FUNCTION_BLOCK ExerciseF_P1
VAR_IN_OUT
	Parameters: GreenMasterBaseParameters;
END_VAR
VAR_INPUT
	EN: BOOL := TRUE;
	ForceExercise: BOOL;
END_VAR
VAR_OUTPUT
	Exercising: BOOL;
END_VAR
VAR
	ExerciseTimer: Timer;
	LocalTime: FB_LocalSystemTime;
	Elapsed: LINT;
	CurrentState: INT;
	StateTimer: TImer;
	DetectedDamperError: BOOL;
	FirstTime: BOOL := TRUE;
END_VAR

LocalTime(bEnable := TRUE);
ExerciseTimer(EN := EN);
Elapsed := ExerciseTimer.ElapsedTime();

StateTimer();
IF EN THEN
	CASE CurrentState OF
		0:
			IF EN AND LocalTime.bValid THEN
				IF ((Parameters.System.Exercise.CirculationPumps.Interval > 0) AND ((ExerciseTimer.ElapsedTime() > (Parameters.System.Exercise.CirculationPumps.Interval * 3600 * 1000)) OR FirstTime) AND 
					(
						(WORD_TO_INT(LocalTime.systemTime.wHour) = Parameters.System.Exercise.CirculationPumps.Hour) AND (WORD_TO_INT(LocalTime.systemTime.wMinute) = Parameters.System.Exercise.CirculationPumps.Minute)
					)) OR ForceExercise THEN
					FirstTime := FALSE;
					ForceExercise := FALSE;
					Exercising := TRUE;
					StateTimer.Restart();
					CurrentState := 1;
					Main.EventLog.LogEvent(EventTypes.Information, 'Exercising P1');
				END_IF			
			END_IF
		1:
			IF StateTimer.ElapsedTime() > 60 * 1000 THEN
				Exercising := FALSE;
				CurrentState := 0;
			END_IF
	END_CASE
END_IF

END_FUNCTION_BLOCK

(* stored: Version 1.1.0.1, ProductVersion 3.1.4024.6
   POU ExerciseF_P1: Id {6854153b-9837-4cc5-be48-d8ec065b240f}, SpecialFunc None *)
